Fanuc KAREL source: kt00258.KL

-- PROVISIONAL review KL for V1013-1; original PC SHA256 3e6f1563558fc8da7a939ec931d26eec8dea0af9a2bca666070b252cb10fd78e
-- Incomplete behavior may be omitted. Consult companion uncertainty JSON. Do not deploy.
PROGRAM KT00258
%NOLOCKGROUP
VAR
  I1 : INTEGER
  R2 : REAL
  OUT : BOOLEAN
BEGIN
  -- UNRESOLVED_PC offsets 5-16; opcodes 2E,23
  -- UNRESOLVED_PC offsets 21-32; opcodes 2E,23
  -- UNRESOLVED_PC offsets 37-58; opcodes 21,21,29,64,6D,23
  -- UNRESOLVED_PC offsets 63-67; opcodes 7F
END KT00258
